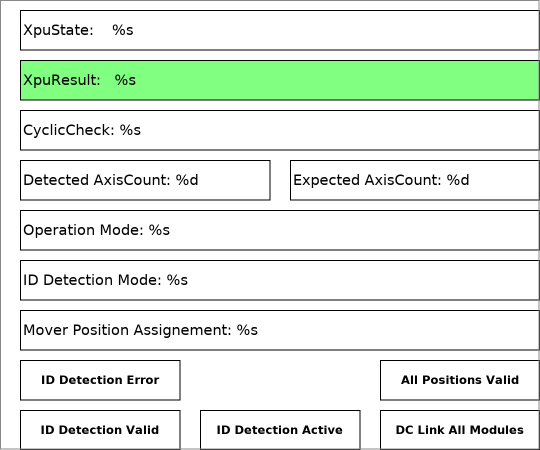
VISUALIZATION XPU_VISU  // 540x450
VAR_IN_OUT
	stXpuState    : ST_XPU_STATE;
  stXpuInfo     : ST_XPU_INFO;
  stXpuStrings  : ST_XPU_STRINGS;
END_VAR
    Rectangle (20,110 520x40), "CyclicCheck: %s", text variable: stXpuStrings.sXpuCyclicCheck
    Rectangle (20,10 520x40), "XpuState: %s", text variable: stXpuStrings.sXpuState
    Rectangle (20,60 520x40), "XpuResult: %s", text variable: stXpuStrings.sXpuResult, colour toggle: (MAIN.eXpuResult = E_PROGRESS.PROGRESS_ERROR)
    Rectangle (380,360 160x40), "All Positions Valid", colour toggle: stXpuInfo.AllPositionsValid
    Rectangle (20,360 160x40), "ID Detection Error", colour toggle: stXpuInfo.IdDetectionError
    Rectangle (20,410 160x40), "ID Detection Valid", colour toggle: stXpuInfo.IdDetectionValid
    Rectangle (200,410 160x40), "ID Detection Active", colour toggle: stXpuInfo.IdDetectionActive
    Rectangle (20,210 520x40), "Operation Mode: %s", text variable: stXpuStrings.sXpuOpMode
    Rectangle (20,260 520x40), "ID Detection Mode: %s", text variable: stXpuStrings.sXpuMoverId_DetectionMode
    Rectangle (20,310 520x40), "Mover Position Assignement: %s", text variable: stXpuStrings.sXpuMoverPosAssignement
    Rectangle (290,160 250x40), "Expected AxisCount: %d", text variable: stXpuInfo.nExpectedAxisCount
    Rectangle (20,160 250x40), "Detected AxisCount: %d", text variable: stXpuInfo.nDetectedAxisCount
    Rectangle (380,410 160x40), "DC Link All Modules", colour toggle: stXpuState.DcLink
END_VISUALIZATION

(* stored: Version 1.1.0.1
   Visu XPU_VISU: Id {39a0c2cb-9f32-46bd-aa63-72985586c43d} *)
